FUNCTION_BLOCK ROBOT_LD90 EXTENDS FB_2_ROB_AMR
VAR_INPUT
	


	sLoadDeliverReturn: Skill_LoadDeliverReturn;
	sEyes: Skill_ROS2_Eyes;
	ComConfig: stComm_TCPIP_Config;
END_VAR
VAR_OUTPUT
  SocketErrorId: UDINT;
END_VAR
VAR
	MissionIndex: INT;
	oldMissionIndex: INT;
	waitTimer: TON;
  COMM: FB_2_Comm_TcpIp;
END_VAR

CYCLIC_AMR();

ComMachine();

//-------- SKILL SETUP ---------


pA_Skills[1]:=ADR(sLoadDeliverReturn);
pA_Skills[2]:=ADR(sEyes);

sEyes();
sLoadDeliverReturn(Rob:=ADR(THIS^));


//------------------------------------

IF MissionIndex<>oldMissionIndex THEN
	waitTimer(IN:=TRUE, PT:=T#4S);
	oldMissionIndex:=MissionIndex;
END_IF
waitTimer();
IF waitTimer.Q THEN
	waitTimer(IN:=FALSE);
	TargetReached:=TRUE;
	ADSLOGSTR(
    msgCtrlMask := ADSLOG_MSGTYPE_HINT,
    msgFmtStr   := 'Simulated target reached!',
    strArg      := ''
);
	
END_IF

METHOD ComMachine : BOOL
VAR_INPUT
END_VAR
// The TCP/IP connection is handled by the communication module.
COMM.Config := ComConfig;
COMM.CYCLIC_TCPIP();

CommunicationReady := COMM.Connected;

bError := COMM.bError;
SocketErrorId := COMM.nErrorId;
nErrorId := TO_UINT(COMM.nErrorId);

ComMachine := NOT bError;
END_METHOD

METHOD Connect : BOOL

Connect := FALSE;

// Validate address
IF LEN(ComConfig.sIpAddress) = 0 THEN
    bError := TRUE;
    RETURN;
END_IF;

// Validate port
IF ComConfig.nPort = 0 THEN
    bError := TRUE;
    RETURN;
END_IF;

// Clear previous error
bError := FALSE;
nErrorId := 0;

Connect := COMM.Connect();
END_METHOD

{warning 'Add property implementation'}
PROPERTY Connected : BOOL
GET
Connected:=COMM.Connected;
END_GET
END_PROPERTY

{warning 'Add method implementation '}
METHOD Disconnect : BOOL
IF COMM.Connected THEN
      Disconnect := TRUE;
      RETURN;
    END_IF

    Disconnect := COMM.Disconnect();
END_METHOD

METHOD PROTECTED OnActivate : eResult
VAR_INPUT
END_VAR

VAR
	eParentResult: eResult;
	myResult: ERESULT;
END_VAR

VAR //YOUR CODE
	succ : BOOL;
END_VAR
eParentResult := SUPER^.OnActivate();
//--------------------------------------------------
myResult:=NONE;
// ----- YOUR CODE HERE (incl. Alarms) -------------

IF bError THEN
    myResult := ERROR;
    ELSIF Connected THEN
      myResult := SUCCESS;
ELSE
      myResult := None;
END_IF

// ----- END YOUR CODE -----------------------------
//--------------------------------------------------
OnActivate := CombineResults(eParentResult,myResult);
END_METHOD

METHOD PROTECTED OnCleanup : eResult
VAR_INPUT
END_VAR

VAR
	eParentResult: eResult;
	myResult: ERESULT;
END_VAR

VAR //YOUR CODE
	succ : BOOL;
END_VAR
eParentResult := SUPER^.OnCleanup();
//--------------------------------------------------
myResult:=NONE;
// ----- YOUR CODE HERE (incl. Alarms) -------------

Disconnect();

    IF COMM.Connected THEN
      myResult := None;
    ELSE
      myResult := SUCCESS;
    END_IF

// ----- END YOUR CODE -----------------------------
//--------------------------------------------------
OnCleanup := CombineResults(eParentResult,myResult);
END_METHOD

METHOD PROTECTED OnConfigure : eResult
VAR_INPUT
END_VAR

VAR
	eParentResult: eResult;
	myResult: ERESULT;
END_VAR

VAR //YOUR CODE
	succ : BOOL;
END_VAR
eParentResult := SUPER^.OnConfigure();
//--------------------------------------------------
myResult:=NONE;
// ----- YOUR CODE HERE (incl. Alarms) -------------

Connect();

    IF bError THEN
      myResult := ERROR;
    ELSIF Connected THEN
      myResult := SUCCESS;
    ELSE
      myResult := None;
    END_IF

// ----- END YOUR CODE -----------------------------
//--------------------------------------------------
OnConfigure := CombineResults(eParentResult,myResult);
END_METHOD

METHOD PROTECTED OnDeactivate : eResult
VAR_INPUT
END_VAR

VAR
	eParentResult: eResult;
	myResult: ERESULT;
END_VAR

VAR //YOUR CODE
	succ : BOOL;
END_VAR
eParentResult := SUPER^.OnDeactivate();
//--------------------------------------------------
myResult:=NONE;
// ----- YOUR CODE HERE (incl. Alarms) -------------

IF bError THEN
    myResult := ERROR;
ELSE
    myResult := SUCCESS;
END_IF

// ----- END YOUR CODE -----------------------------
//--------------------------------------------------
OnDeactivate := CombineResults(eParentResult,myResult);
END_METHOD

METHOD PROTECTED OnError : eResult
VAR_INPUT
END_VAR

VAR
	eParentResult: eResult;
	myResult: ERESULT;
END_VAR

VAR //YOUR CODE
	succ : BOOL;
END_VAR
eParentResult := SUPER^.OnError();
//--------------------------------------------------
myResult:=NONE;
// ----- YOUR CODE HERE (incl. Alarms) -------------

myResult := SUCCESS;

// ----- END YOUR CODE -----------------------------
//--------------------------------------------------
OnError := CombineResults(eParentResult,myResult);
END_METHOD

METHOD PROTECTED OnShutdown : eResult
VAR_INPUT
END_VAR

VAR
	eParentResult: eResult;
	myResult: ERESULT;
END_VAR

VAR //YOUR CODE
	succ : BOOL;
END_VAR
eParentResult := SUPER^.OnShutdown();
//--------------------------------------------------
myResult:=NONE;
// ----- YOUR CODE HERE (incl. Alarms) -------------

Disconnect();

    IF COMM.Connected THEN
      myResult := None;
    ELSIF bError THEN
      myResult := ERROR;
    ELSE
      myResult := SUCCESS;
    END_IF

// ----- END YOUR CODE -----------------------------
//--------------------------------------------------
OnShutdown := CombineResults(eParentResult,myResult);
END_METHOD

METHOD ResetConnection : BOOL
bError := FALSE;
nErrorId := 0;
SocketErrorId := 0;

COMM.Reset();
ResetConnection := COMM.Reconnect();
END_METHOD

END_FUNCTION_BLOCK

(* stored: Version 1.1.0.1, ProductVersion 3.1.4026.18
   POU ROBOT_LD90: Id {fac74160-c2b3-4f77-bd69-eddf1970c653}, SpecialFunc None
   Folder Communication: Id {2a9c337e-719c-4121-a5a9-4ddfd8584a43}
   Folder StateControl: Id {67994def-610e-4a0b-a6c8-85df31e22884}
   Method ComMachine: Id {040d86b8-c78e-42d4-a5c1-25c0270b6e14}
   Method Connect: Id {70fa978a-67c6-43be-99fb-d03c8689cf07}
   Property Connected: Id {e71d8962-d52b-46f4-b79d-88e001b39f65}
   Get Get: Id {1724321d-02c7-40cd-942a-414eba41ba06}
   Method Disconnect: Id {c75c2374-9ebb-4dd8-a5bc-f61f0a69c931}
   Method OnActivate: Id {7fa92802-2ede-4193-9973-ad7754d17239}
   Method OnCleanup: Id {7747948a-f8e1-4cdb-8a20-610ab536a0ef}
   Method OnConfigure: Id {c568c508-6321-435c-b7c4-683ad73a8f42}
   Method OnDeactivate: Id {57ce1156-6b80-40b7-8fff-100660e6e779}
   Method OnError: Id {74c0a508-94ea-4785-a0ea-1af2639ff5e5}
   Method OnShutdown: Id {f496723a-9c1c-413c-b4ed-4d78c56c0863}
   Method ResetConnection: Id {1a6fc39d-923f-4cb8-bc55-cd413f8ec29d} *)
